(* PLC project Laboratorio 2, Desconocido Embaladora 1 *)
(* stored: creationDateTime 2022-10-29T15:41:28, modificationDateTime 2022-10-31T23:03:56 *)

PROGRAM program0
  VAR
    Joysick AT %IW0 : INT := 512;  (* Representa el joystick, toma los valores que se leen. *)
  END_VAR
  VAR
    ValAv : INT := 700;  (* Valor del joystick para que gire a sentido horario *)
    ValRet : INT := 300;  (* Valor del joystick para que gire a sentido antihorario *)
  END_VAR
  VAR
    BobinaA AT %QX0.3 : BOOL := 0;
    BobinaB AT %QX0.1 : BOOL := 0;
    BobinaC AT %QX0.0 : BOOL := 0;
    BobinaD AT %QX0.2 : BOOL := 0;
  END_VAR
  VAR
    Reloj : TIME := T#200ms;  (* Duración del paso *)
    RelojA : TIME := T#0ms;  (* Paso para la bobina A *)
    RelojB : TIME := T#200ms;  (* Paso para la bobina B *)
    RelojC : TIME := T#400ms;  (* Paso para la bobina C *)
    RelojD : TIME := T#600ms;  (* Paso para la bobina D *)
    Clock : TIME := T#1s400ms;  (* Pasos *)
    TON0 : TON;
    TON1 : TON;
    TP0 : TP;
    TP1 : TP;
    TON2 : TON;
    TP2 : TP;
    TON3 : TON;
    TP3 : TP;
    TON4 : TON;
    TP4 : TP;
  END_VAR
  VAR  (* added by the conversion: wires and edge detectors of the diagram *)
    _AND45_OUT : BOOL;
    _LE16_OUT : BOOL;
  END_VAR

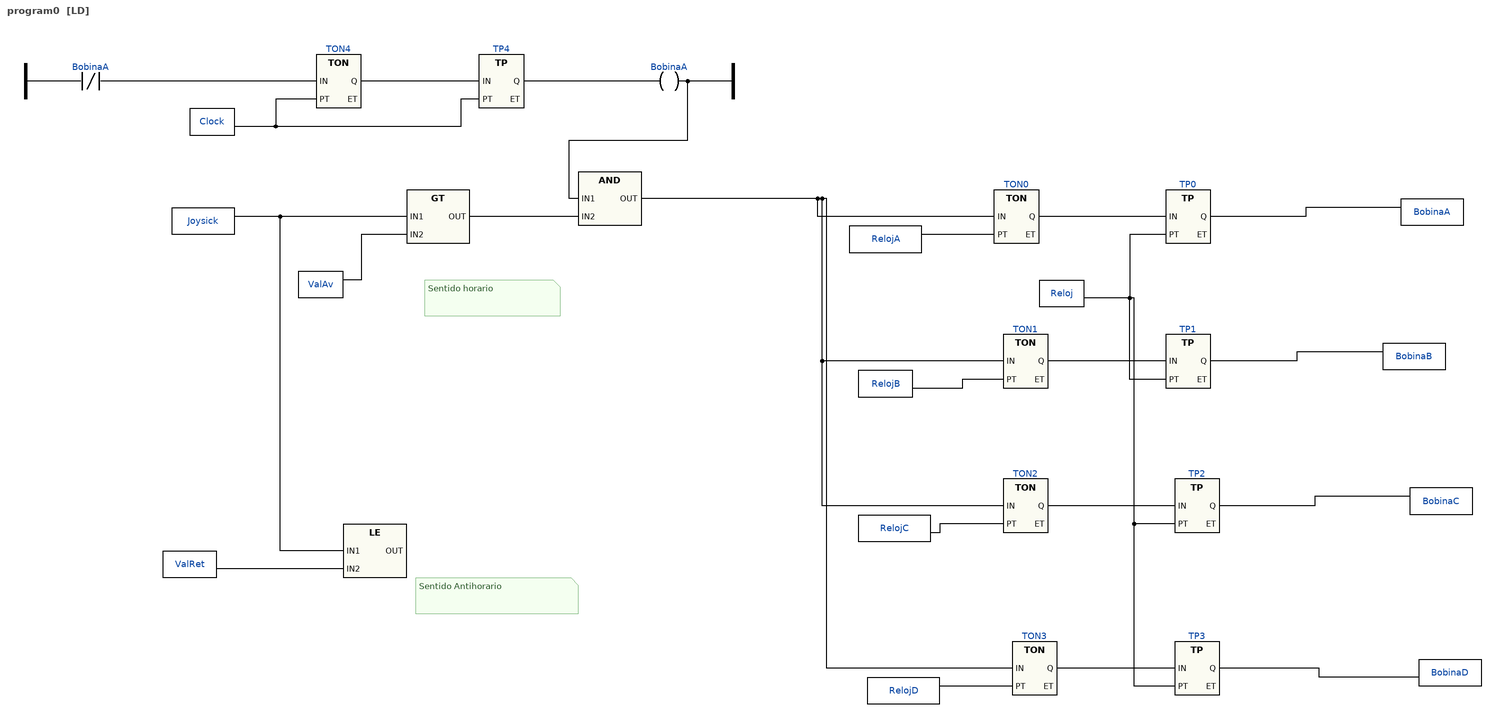
(* LD diagram, written out as Structured Text *)
TON4(IN := NOT BobinaA, PT := Clock);
TP4(IN := TON4.Q, PT := Clock);
BobinaA := TP4.Q;
_AND45_OUT := TP4.Q AND Joysick > ValAv;
TON0(IN := _AND45_OUT, PT := RelojA);
TP0(IN := TON0.Q, PT := Reloj);
BobinaA := TP0.Q;
(* Sentido horario *)
TON1(IN := _AND45_OUT, PT := RelojB);
TP1(IN := TON1.Q, PT := Reloj);
BobinaB := TP1.Q;
TON2(IN := _AND45_OUT, PT := RelojC);
TP2(IN := TON2.Q, PT := Reloj);
BobinaC := TP2.Q;
(* Sentido Antihorario *)
TON3(IN := _AND45_OUT, PT := RelojD);
TP3(IN := TON3.Q, PT := Reloj);
BobinaD := TP3.Q;
_LE16_OUT := Joysick <= ValRet;
END_PROGRAM

CONFIGURATION Config0
  RESOURCE Res0 ON PLC
    TASK task0(INTERVAL := T#20ms, PRIORITY := 0);
    PROGRAM instance0 WITH task0 : program0;
  END_RESOURCE
END_CONFIGURATION
